// TIA Portal V20 export
TYPE "UDT_EstadoZonaDispositivo"
   STRUCT
      Pulsador { S7_SetPoint := 'True'} : "PulsadorZona";
      Estado { S7_SetPoint := 'True'} : "EstadoZona";   // Estado de la Zona
      CodigoError : UDInt;   // Codigo de Error de la Zona
      VariablesInternas { S7_SetPoint := 'True'} : "InternasDeLaZona";   // Variables internas y sinoptico
   END_STRUCT;
   // Pulsador.P_Auto := false;
END_TYPE
